Omron CX-Programmer project 新工程 (CX-Programmer 9.50)

# PLC 新PLC1: CP1H XA

## Global symbols (name address type ; comment)
0.01 BOOL  ; 启动
0.02 BOOL  ; 停止
0.04 BOOL  ; 急停
0.05 BOOL  ; 相序保护
0.11 BOOL  ; 空压机热保护
100.03 BOOL  ; A平
100.04 BOOL  ; B平
100.05 BOOL  ; C平
100.06 BOOL  ; A进
100.07 BOOL  ; B进
101.00 BOOL  ; C进
101.01 BOOL  ; A排
101.02 BOOL  ; b排
101.03 BOOL  ; C排
10.00 BOOL  ; 连续与自动
200 CHANNEL  ; 氧气纯度
201 CHANNEL  ; 空气压力
202 CHANNEL  ; 氧气压力
203 CHANNEL  ; 露点
A526.01 BOOL  ; 串行端口1重启标志
A528.11 BOOL  ; 出错标志
D1 CHANNEL  ; 空气压力上限
D10 CHANNEL  ; 屏显露点
D11 CHANNEL  ; 屏显氧气压力
D12 CHANNEL  ; 屏输空气压力下限
D13 CHANNEL  ; 屏显油温
D15 CHANNEL  ; 屏输空气压力上限
D17 CHANNEL  ; 屏输空气压力下限
D19 CHANNEL  ; 屏输氧气压力上限
D2 CHANNEL  ; 空气压力下限
D20 CHANNEL  ; 制氧机工作状态
D21 CHANNEL  ; 屏输氧气压力下限
D3 CHANNEL  ; 氧气压力上限
D3102 CHANNEL  ; 流量高位
D3103 CHANNEL  ; 流量低位
D3104 CHANNEL  ; 总流量高位
D3105 CHANNEL  ; 总流量低位
D317 CHANNEL  ; 制氧机状态字
D318 CHANNEL  ; 冷干机状态字
D321 CHANNEL  ; 系统状态字
D331 CHANNEL  ; 空压机状态字
D332 CHANNEL  ; 空滤维保计时
D333 CHANNEL  ; 油滤维保计时
D334 CHANNEL  ; 油分维保计时
D335 CHANNEL  ; 机油维保计时
D336 CHANNEL  ; 管滤维保计时
D337 CHANNEL  ; 菌滤维保计时
D338 CHANNEL  ; 制氧机工作状态
D4 CHANNEL  ; 氧气压力下限
D50 CHANNEL  ; 瞬时流量
D51 CHANNEL  ; 瞬时流量
D65 CHANNEL  ; 氧气压力
D66 CHANNEL  ; 空气压力
D67 CHANNEL  ; 油温
D68 CHANNEL  ; 氧气纯度
D69 CHANNEL  ; 氧气流量
D7 CHANNEL  ; 屏显氧气纯度
D8 CHANNEL  ; 屏显空气压力
D80 CHANNEL  ; 远程氧气
D82 CHANNEL  ; 远程空气
D84 CHANNEL  ; 远程油温
D86 CHANNEL  ; 远程氧气纯度
D88 CHANNEL  ; 远程氧气流量
D9 CHANNEL  ; 屏显空气压力
H1 CHANNEL  ; 运行总时间
H10.00 BOOL  ; 远程控制停机（保持）
H2 CHANNEL  ; 空滤维保计时
H3 CHANNEL  ; 油滤维保计时
H4 CHANNEL  ; 油分维保计时
H5 CHANNEL  ; 机油维保计时
H6 CHANNEL  ; 管滤维保计时
H7 CHANNEL  ; 菌滤维保计时
T0200 BOOL  ; 产生0.2秒脉冲
W10.00 BOOL  ; 连续与自动
W21.00 BOOL  ; 启动标志1
W21.01 BOOL  ; 散热见机
W21.02 BOOL  ; 外接排风
W21.03 BOOL  ; 冷干机
W21.04 BOOL  ; 卸载电磁阀
W21.05 BOOL  ; 空压机
W21.06 BOOL  ; 油温开关
W21.08 BOOL  ; 运行标志
W21.09 BOOL  ; 停机保护2分钟
W21.10 BOOL  ; 启动标志2
W21.11 BOOL  ; 出氧电磁阀
W21.12 BOOL  ; 准备待机
W21.13 BOOL  ; 待机
W21.14 BOOL  ; 复位几个启动时间
W21.15 BOOL  ; 解除几个停机时间
W22.01 BOOL  ; 连续与自动
W22.06 BOOL  ; 油温开关
W23.00 BOOL  ; 制氧启动最低空气压力
W24.01 BOOL  ; 准备停机
W24.07 BOOL  ; 停机
W25.00 BOOL  ; 报警器
W30 CHANNEL  ; 屏显氧气纯度
W32.00 BOOL  ; 散热风机热保护
W32.01 BOOL  ; 报警解除
W50.01 BOOL  ; 空滤维保复位
W50.02 BOOL  ; 油滤维保复位
W50.03 BOOL  ; 油分维保复位
W50.04 BOOL  ; 机油维保复位
W50.05 BOOL  ; 管滤维保复位
W50.06 BOOL  ; 菌滤维保复位
W50.15 BOOL  ; 躲开开机时氧气压力低
W8 CHANNEL  ; 计数器值

## Program 新程序1 (cyclic task 0)
Local symbols
Dd112 UINT
Dd300 UINT_BCD
P_0_6s BOOL
P_2分钟 BOOL
P_30分钟 BOOL
W BOOL
b189 UINT
ffff UINT

### Section 启动停止

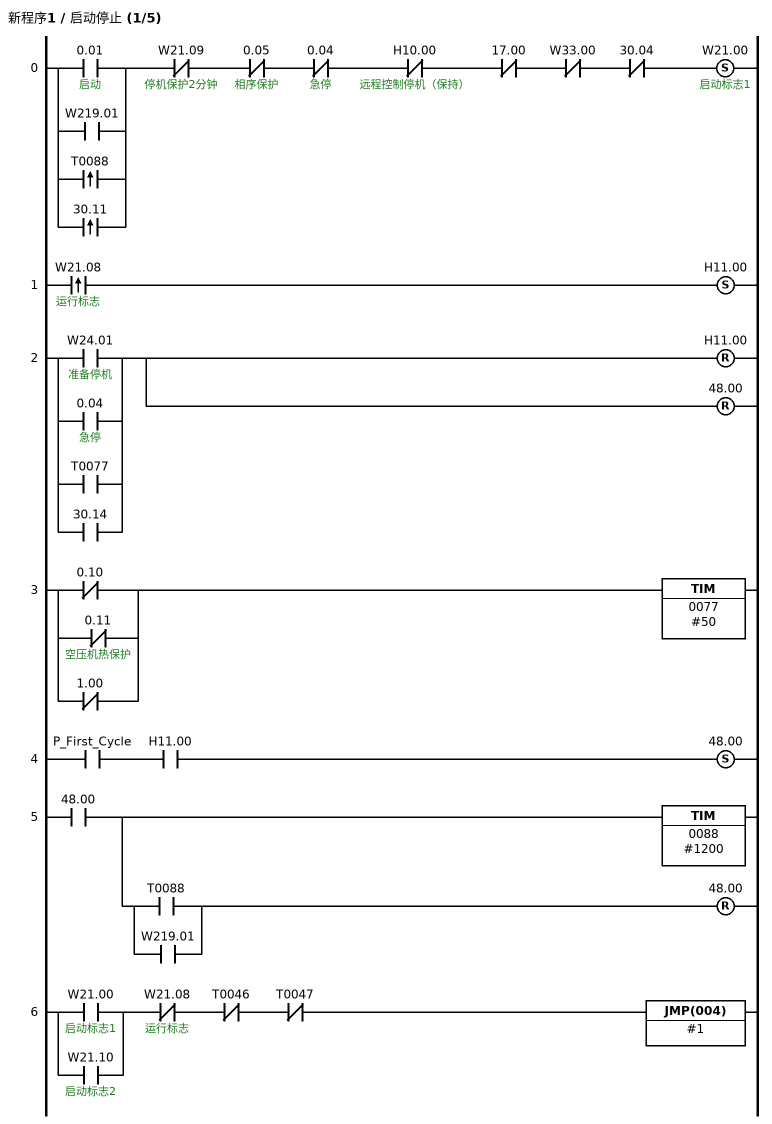
; rung 0
LD 0.01  ; 启动
OR W219.01
@OR T0088
@OR 30.11
ANDNOT W21.09  ; 停机保护2分钟
ANDNOT 0.05  ; 相序保护
ANDNOT 0.04  ; 急停
ANDNOT H10.00  ; 远程控制停机（保持）
ANDNOT 17.00
ANDNOT W33.00
ANDNOT 30.04
SET W21.00  ; 启动标志1
; rung 1
@LD W21.08  ; 运行标志
SET H11.00
; rung 2
LD W24.01  ; 准备停机
OR 0.04  ; 急停
OR T0077
OR 30.14
RSET H11.00
RSET 48.00
; rung 3
LDNOT 0.10
ORNOT 0.11  ; 空压机热保护
ORNOT 1.00
TIM 0077 #50
; rung 4
LD P_First_Cycle
AND H11.00
SET 48.00
; rung 5
LD 48.00
TIM 0088 #1200
LD T0088
OR W219.01
ANDLD
RSET 48.00
; rung 6
LD W21.00  ; 启动标志1
OR W21.10  ; 启动标志2
ANDNOT W21.08  ; 运行标志
ANDNOT T0046
ANDNOT T0047
JMP(004) #1

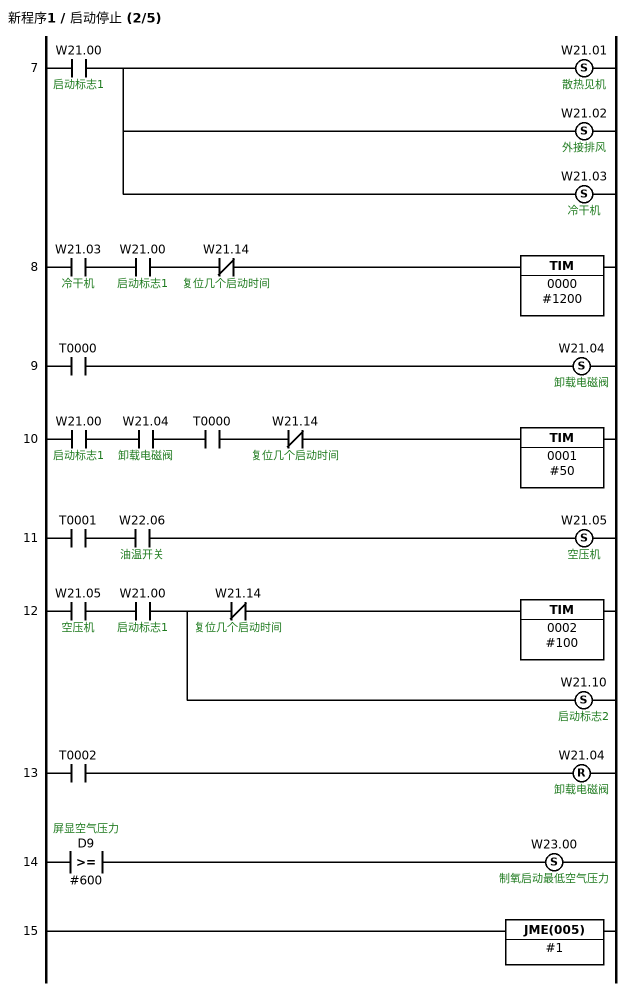
; rung 7
LD W21.00  ; 启动标志1
SET W21.01  ; 散热见机
SET W21.02  ; 外接排风
SET W21.03  ; 冷干机
; rung 8
LD W21.03  ; 冷干机
AND W21.00  ; 启动标志1
ANDNOT W21.14  ; 复位几个启动时间
TIM 0000 #1200
; rung 9
LD T0000
SET W21.04  ; 卸载电磁阀
; rung 10
LD W21.00  ; 启动标志1
AND W21.04  ; 卸载电磁阀
AND T0000
ANDNOT W21.14  ; 复位几个启动时间
TIM 0001 #50
; rung 11
LD T0001
AND W22.06  ; 油温开关
SET W21.05  ; 空压机
; rung 12
LD W21.05  ; 空压机
AND W21.00  ; 启动标志1
OUT TR0
ANDNOT W21.14  ; 复位几个启动时间
TIM 0002 #100
LD TR0
SET W21.10  ; 启动标志2
; rung 13
LD T0002
RSET W21.04  ; 卸载电磁阀
; rung 14
LD>=(325) D9 #600  ; 屏显空气压力
SET W23.00  ; 制氧启动最低空气压力
; rung 15
JME(005) #1

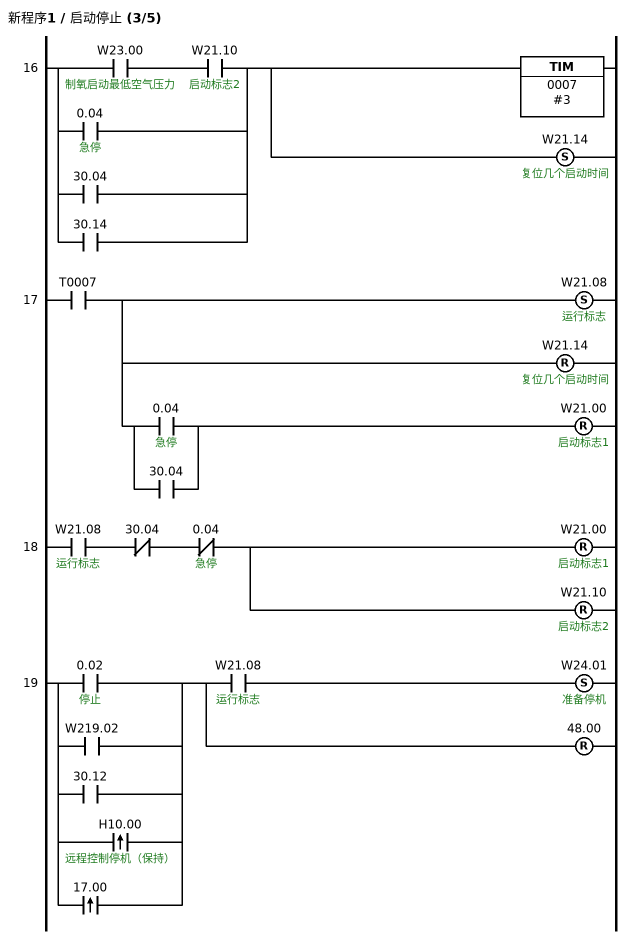
; rung 16
LD W23.00  ; 制氧启动最低空气压力
AND W21.10  ; 启动标志2
OR 0.04  ; 急停
OR 30.04
OR 30.14
TIM 0007 #3
SET W21.14  ; 复位几个启动时间
; rung 17
LD T0007
SET W21.08  ; 运行标志
RSET W21.14  ; 复位几个启动时间
LD 0.04  ; 急停
OR 30.04
ANDLD
RSET W21.00  ; 启动标志1
; rung 18
LD W21.08  ; 运行标志
ANDNOT 30.04
ANDNOT 0.04  ; 急停
RSET W21.00  ; 启动标志1
RSET W21.10  ; 启动标志2
; rung 19
LD 0.02  ; 停止
OR W219.02
OR 30.12
@OR H10.00  ; 远程控制停机（保持）
@OR 17.00
OUT TR0
AND W21.08  ; 运行标志
SET W24.01  ; 准备停机
LD TR0
RSET 48.00

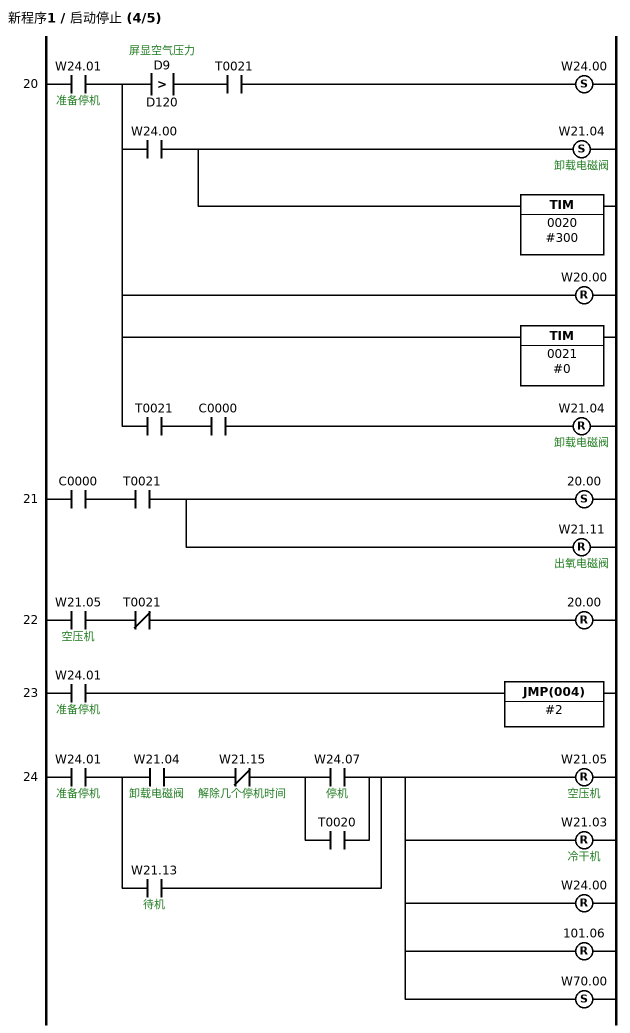
; rung 20
LD W24.01  ; 准备停机
OUT TR0
AND>(320) D9 D120  ; 屏显空气压力
AND T0021
SET W24.00
LD TR0
AND W24.00
SET W21.04  ; 卸载电磁阀
TIM 0020 #300
LD TR0
RSET W20.00
TIM 0021 #0
AND T0021
AND C0000
RSET W21.04  ; 卸载电磁阀
; rung 21
LD C0000
AND T0021
SET 20.00
RSET W21.11  ; 出氧电磁阀
; rung 22
LD W21.05  ; 空压机
ANDNOT T0021
RSET 20.00
; rung 23
LD W24.01  ; 准备停机
JMP(004) #2
; rung 24
LD W24.01  ; 准备停机
LD W21.04  ; 卸载电磁阀
ANDNOT W21.15  ; 解除几个停机时间
LD W24.07  ; 停机
OR T0020
ANDLD
OR W21.13  ; 待机
ANDLD
RSET W21.05  ; 空压机
RSET W21.03  ; 冷干机
RSET W24.00
RSET 101.06
SET W70.00

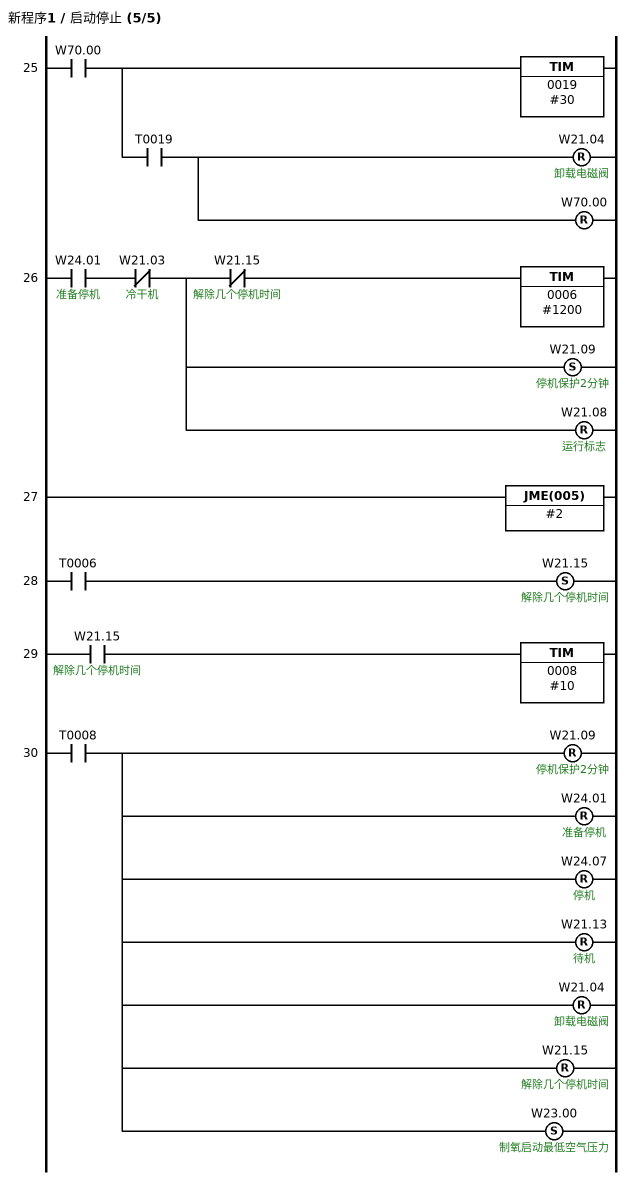
; rung 25
LD W70.00
TIM 0019 #30
AND T0019
RSET W21.04  ; 卸载电磁阀
RSET W70.00
; rung 26
LD W24.01  ; 准备停机
ANDNOT W21.03  ; 冷干机
OUT TR0
ANDNOT W21.15  ; 解除几个停机时间
TIM 0006 #1200
LD TR0
SET W21.09  ; 停机保护2分钟
RSET W21.08  ; 运行标志
; rung 27
JME(005) #2
; rung 28
LD T0006
SET W21.15  ; 解除几个停机时间
; rung 29
LD W21.15  ; 解除几个停机时间
TIM 0008 #10
; rung 30
LD T0008
RSET W21.09  ; 停机保护2分钟
RSET W24.01  ; 准备停机
RSET W24.07  ; 停机
RSET W21.13  ; 待机
RSET W21.04  ; 卸载电磁阀
RSET W21.15  ; 解除几个停机时间
SET W23.00  ; 制氧启动最低空气压力

### Section 制氧机时间

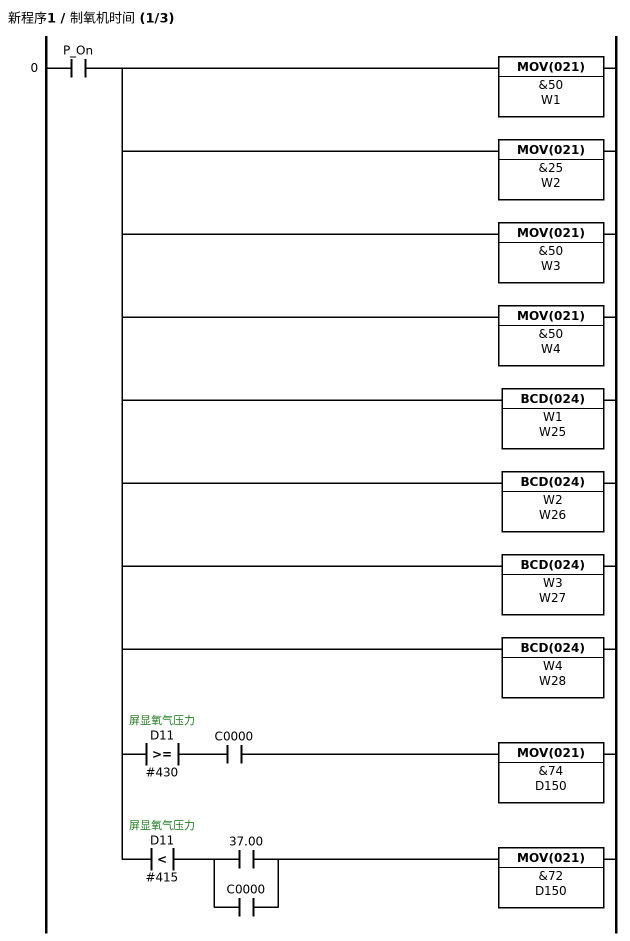
; rung 0
LD P_On
OUT TR0
MOV(021) &50 W1
MOV(021) &25 W2
MOV(021) &50 W3
MOV(021) &50 W4
BCD(024) W1 W25
BCD(024) W2 W26
BCD(024) W3 W27
BCD(024) W4 W28
AND>=(325) D11 #430  ; 屏显氧气压力
AND C0000
MOV(021) &74 D150
LD TR0
AND<(310) D11 #415  ; 屏显氧气压力
LD 37.00
OR C0000
ANDLD
MOV(021) &72 D150

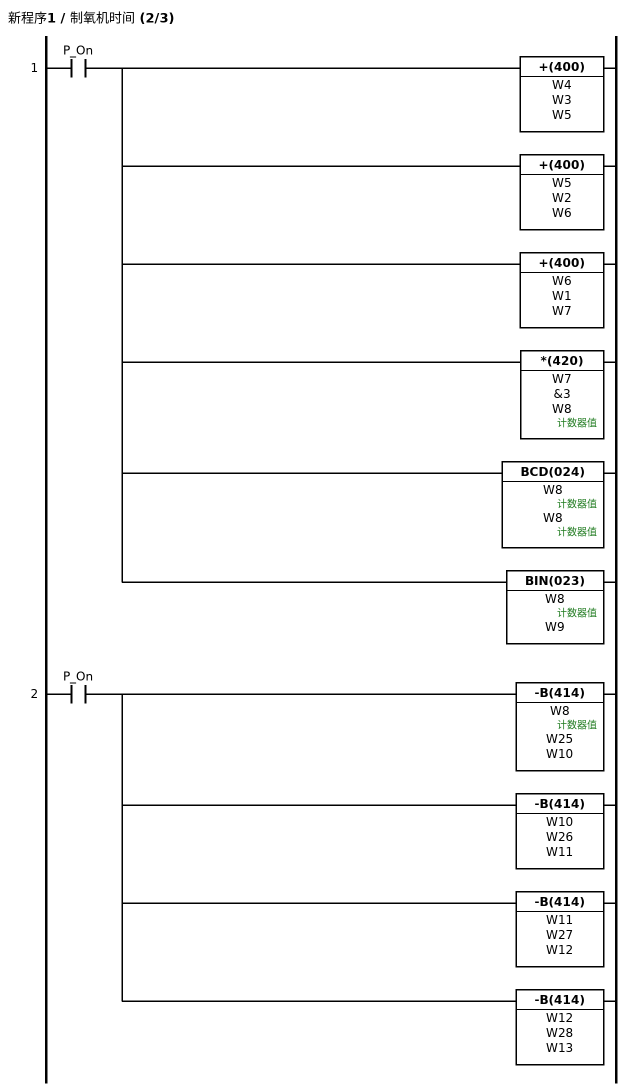
; rung 1
LD P_On
+(400) W4 W3 W5
+(400) W5 W2 W6
+(400) W6 W1 W7
*(420) W7 &3 W8  ; 计数器值
BCD(024) W8 W8  ; 计数器值
BIN(023) W8 W9  ; 计数器值
; rung 2
LD P_On
-B(414) W8 W25 W10  ; 计数器值
-B(414) W10 W26 W11
-B(414) W11 W27 W12
-B(414) W12 W28 W13

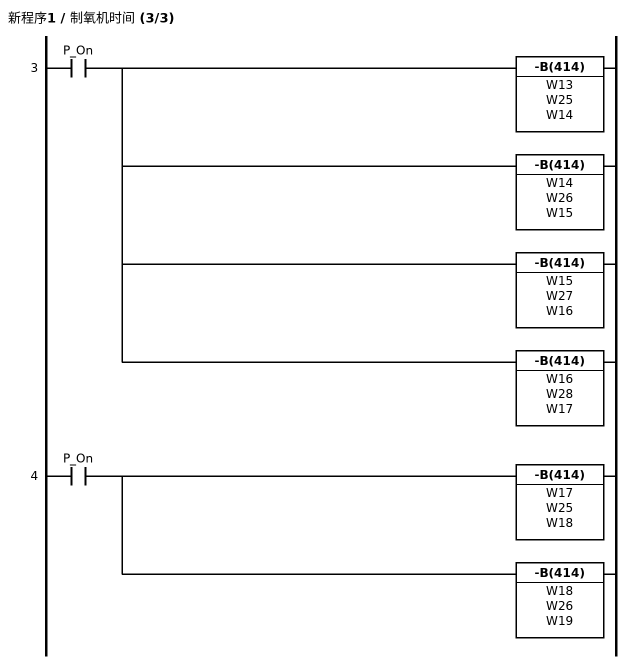
; rung 3
LD P_On
-B(414) W13 W25 W14
-B(414) W14 W26 W15
-B(414) W15 W27 W16
-B(414) W16 W28 W17
; rung 4
LD P_On
-B(414) W17 W25 W18
-B(414) W18 W26 W19

### Section 制氧机步骤

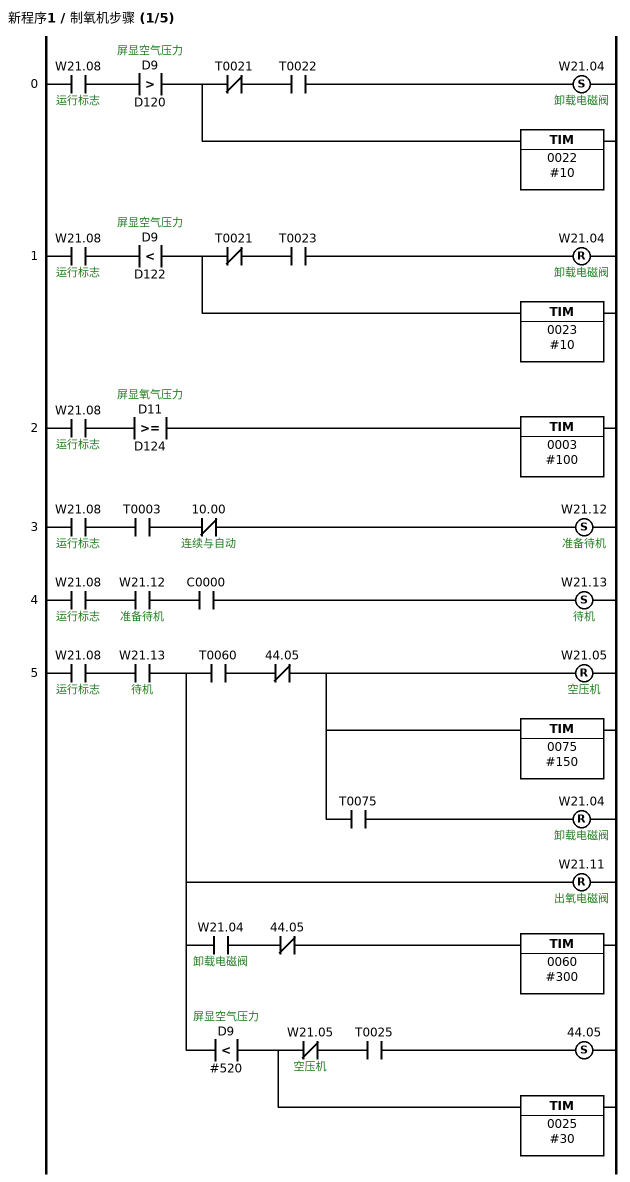
; rung 0
LD W21.08  ; 运行标志
AND>(320) D9 D120  ; 屏显空气压力
OUT TR0
ANDNOT T0021
AND T0022
SET W21.04  ; 卸载电磁阀
LD TR0
TIM 0022 #10
; rung 1
LD W21.08  ; 运行标志
AND<(310) D9 D122  ; 屏显空气压力
OUT TR0
ANDNOT T0021
AND T0023
RSET W21.04  ; 卸载电磁阀
LD TR0
TIM 0023 #10
; rung 2
LD W21.08  ; 运行标志
AND>=(325) D11 D124  ; 屏显氧气压力
TIM 0003 #100
; rung 3
LD W21.08  ; 运行标志
AND T0003
ANDNOT 10.00  ; 连续与自动
SET W21.12  ; 准备待机
; rung 4
LD W21.08  ; 运行标志
AND W21.12  ; 准备待机
AND C0000
SET W21.13  ; 待机
; rung 5
LD W21.08  ; 运行标志
AND W21.13  ; 待机
OUT TR0
AND T0060
ANDNOT 44.05
RSET W21.05  ; 空压机
TIM 0075 #150
AND T0075
RSET W21.04  ; 卸载电磁阀
LD TR0
RSET W21.11  ; 出氧电磁阀
AND W21.04  ; 卸载电磁阀
ANDNOT 44.05
TIM 0060 #300
LD TR0
AND<(310) D9 #520  ; 屏显空气压力
OUT TR0
ANDNOT W21.05  ; 空压机
AND T0025
SET 44.05
LD TR0
TIM 0025 #30

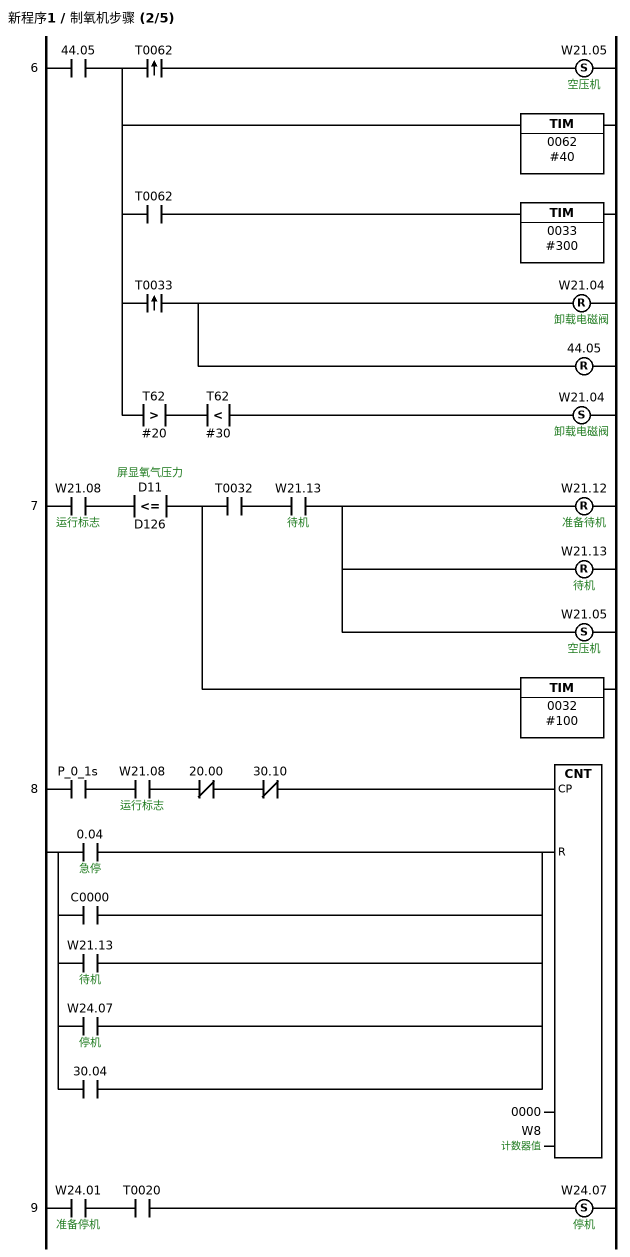
; rung 6
LD 44.05
OUT TR0
@AND T0062
SET W21.05  ; 空压机
LD TR0
TIM 0062 #40
AND T0062
TIM 0033 #300
LD TR0
@AND T0033
RSET W21.04  ; 卸载电磁阀
RSET 44.05
LD TR0
AND>(320) T62 #20
AND<(310) T62 #30
SET W21.04  ; 卸载电磁阀
; rung 7
LD W21.08  ; 运行标志
AND<=(315) D11 D126  ; 屏显氧气压力
OUT TR0
AND T0032
AND W21.13  ; 待机
RSET W21.12  ; 准备待机
RSET W21.13  ; 待机
SET W21.05  ; 空压机
LD TR0
TIM 0032 #100
; rung 8
LD P_0_1s
AND W21.08  ; 运行标志
ANDNOT 20.00
ANDNOT 30.10
LD 0.04  ; 急停
OR C0000
OR W21.13  ; 待机
OR W24.07  ; 停机
OR 30.04
CNT 0000 W8  ; 计数器值
; rung 9
LD W24.01  ; 准备停机
AND T0020
SET W24.07  ; 停机

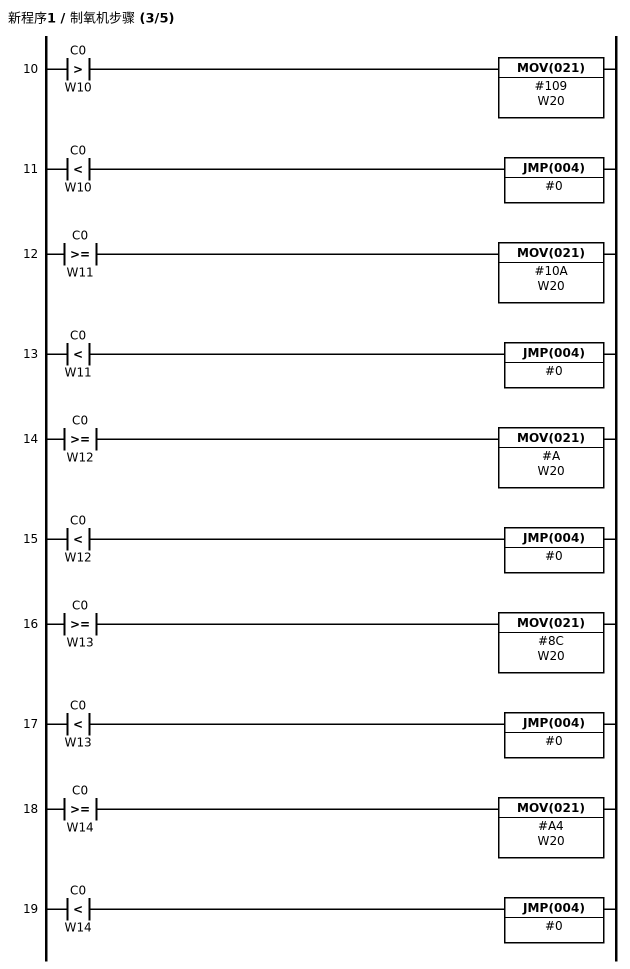
; rung 10
LD>(320) C0 W10
MOV(021) #109 W20
; rung 11
LD<(310) C0 W10
JMP(004) #0
; rung 12
LD>=(325) C0 W11
MOV(021) #10A W20
; rung 13
LD<(310) C0 W11
JMP(004) #0
; rung 14
LD>=(325) C0 W12
MOV(021) #A W20
; rung 15
LD<(310) C0 W12
JMP(004) #0
; rung 16
LD>=(325) C0 W13
MOV(021) #8C W20
; rung 17
LD<(310) C0 W13
JMP(004) #0
; rung 18
LD>=(325) C0 W14
MOV(021) #A4 W20
; rung 19
LD<(310) C0 W14
JMP(004) #0

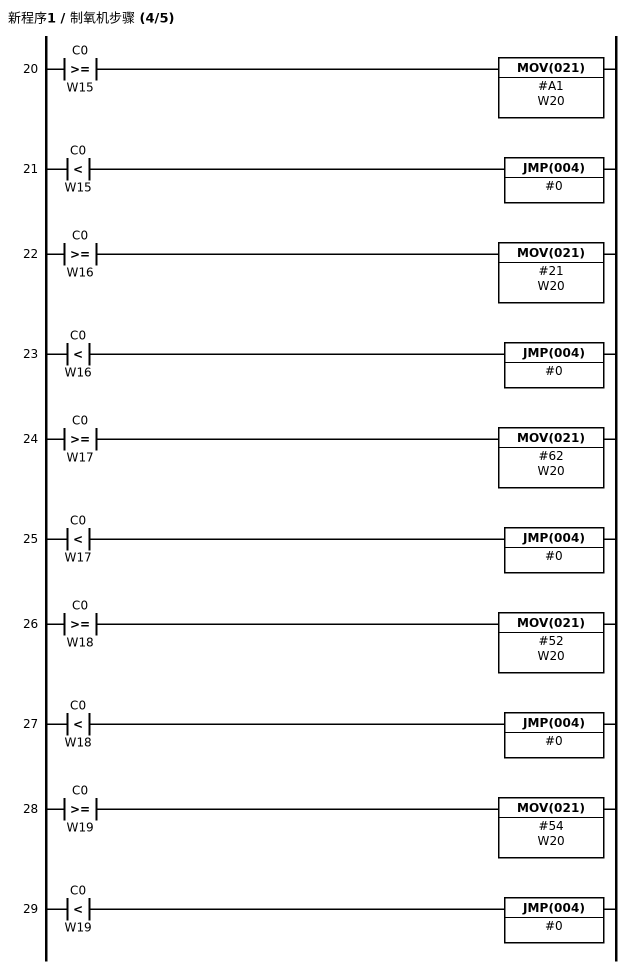
; rung 20
LD>=(325) C0 W15
MOV(021) #A1 W20
; rung 21
LD<(310) C0 W15
JMP(004) #0
; rung 22
LD>=(325) C0 W16
MOV(021) #21 W20
; rung 23
LD<(310) C0 W16
JMP(004) #0
; rung 24
LD>=(325) C0 W17
MOV(021) #62 W20
; rung 25
LD<(310) C0 W17
JMP(004) #0
; rung 26
LD>=(325) C0 W18
MOV(021) #52 W20
; rung 27
LD<(310) C0 W18
JMP(004) #0
; rung 28
LD>=(325) C0 W19
MOV(021) #54 W20
; rung 29
LD<(310) C0 W19
JMP(004) #0

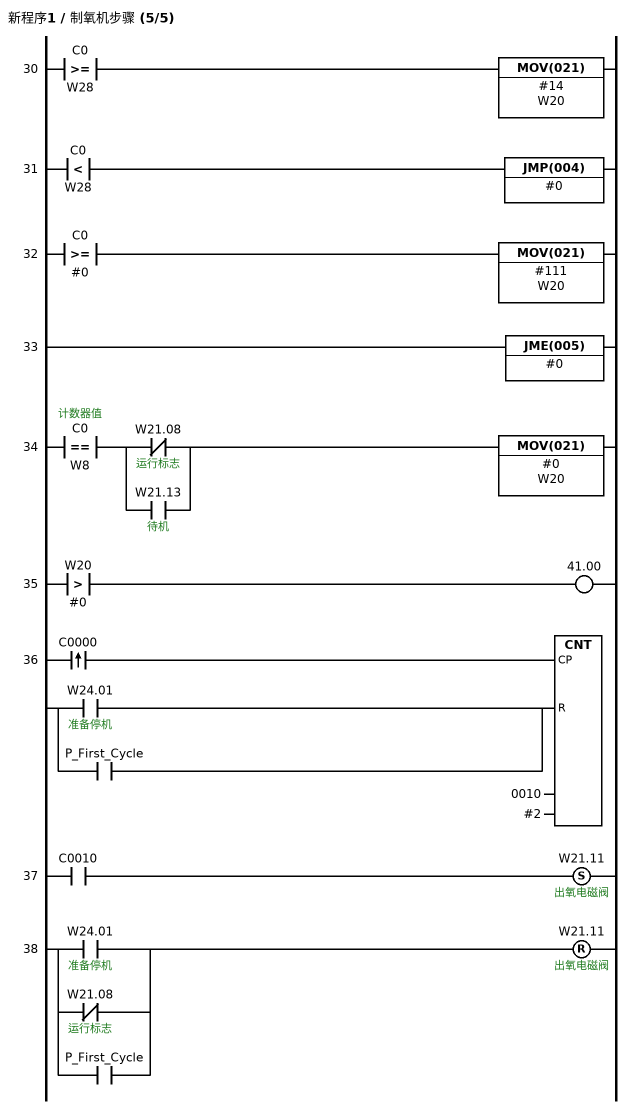
; rung 30
LD>=(325) C0 W28
MOV(021) #14 W20
; rung 31
LD<(310) C0 W28
JMP(004) #0
; rung 32
LD>=(325) C0 #0
MOV(021) #111 W20
; rung 33
JME(005) #0
; rung 34
LD=(300) C0 W8  ; 计数器值
LDNOT W21.08  ; 运行标志
OR W21.13  ; 待机
ANDLD
MOV(021) #0 W20
; rung 35
LD>(320) W20 #0
OUT 41.00
; rung 36
@LD C0000
LD W24.01  ; 准备停机
OR P_First_Cycle
CNT 0010 #2
; rung 37
LD C0010
SET W21.11  ; 出氧电磁阀
; rung 38
LD W24.01  ; 准备停机
ORNOT W21.08  ; 运行标志
OR P_First_Cycle
RSET W21.11  ; 出氧电磁阀

### Section _4AD数值

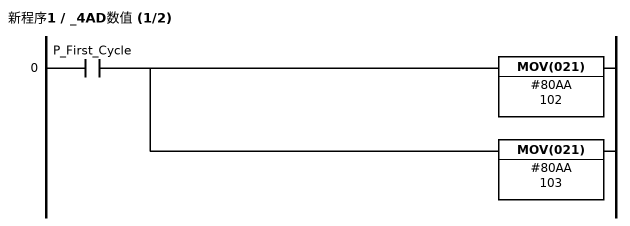
; rung 0
LD P_First_Cycle
MOV(021) #80AA 102
MOV(021) #80AA 103

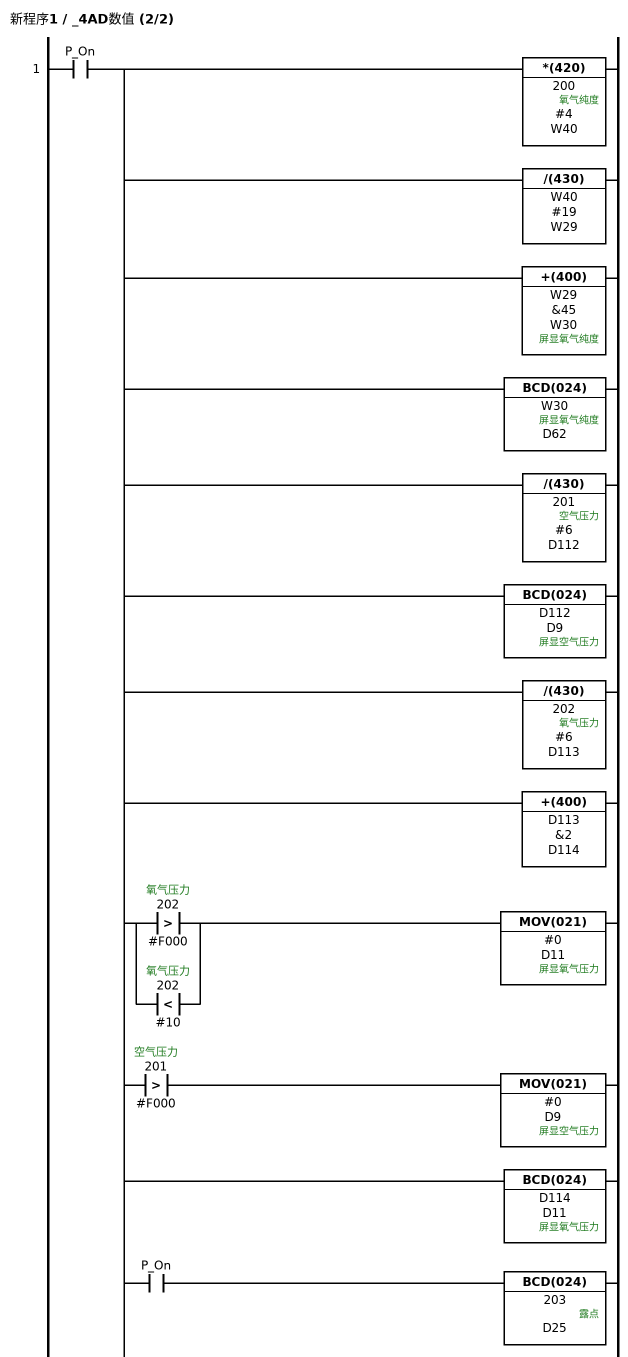

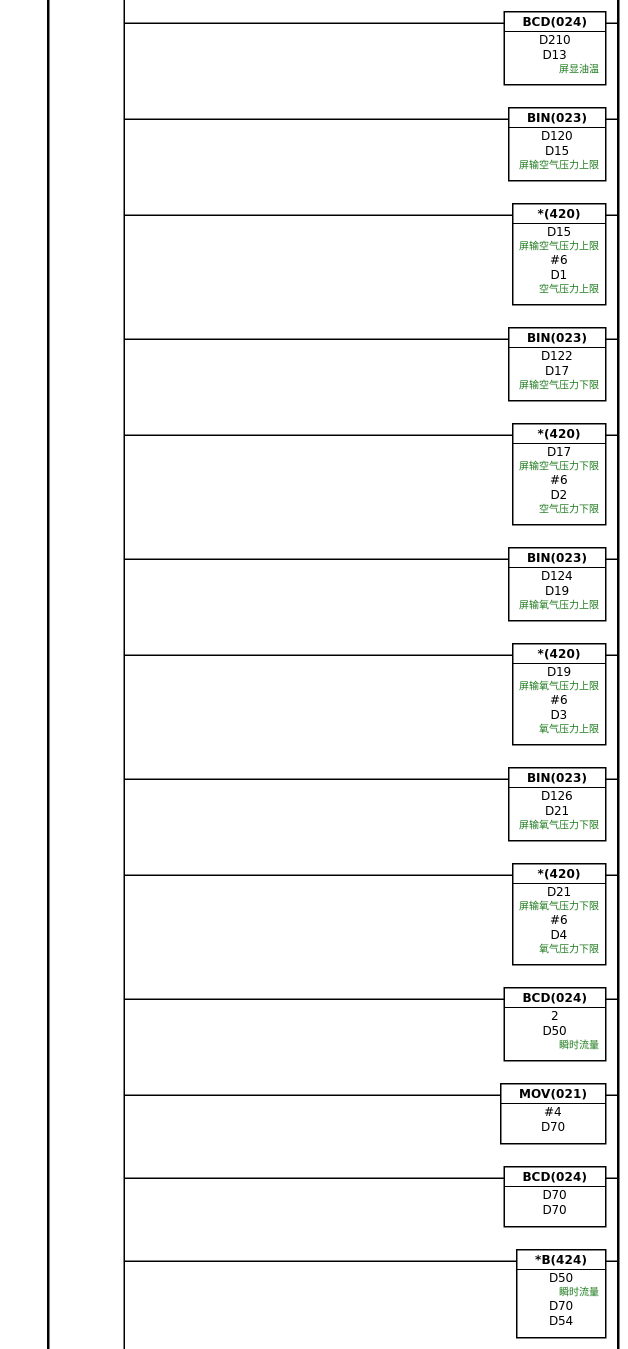

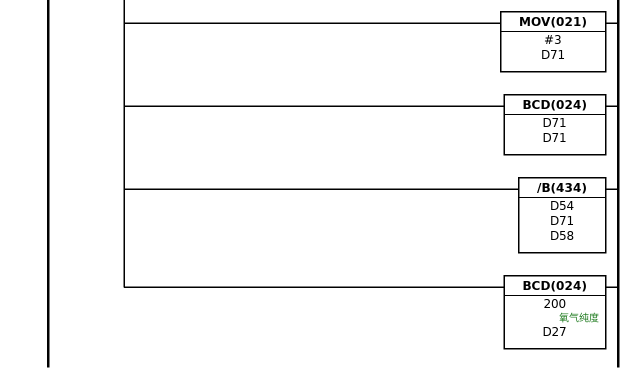
; rung 1
LD P_On
OUT TR0
*(420) 200 #4 W40  ; 氧气纯度
/(430) W40 #19 W29
+(400) W29 &45 W30  ; 屏显氧气纯度
BCD(024) W30 D62  ; 屏显氧气纯度
/(430) 201 #6 D112  ; 空气压力
BCD(024) D112 D9  ; 屏显空气压力
/(430) 202 #6 D113  ; 氧气压力
+(400) D113 &2 D114
LD>(320) 202 #F000  ; 氧气压力
OR<(310) 202 #10  ; 氧气压力
ANDLD
MOV(021) #0 D11  ; 屏显氧气压力
LD TR0
AND>(320) 201 #F000  ; 空气压力
MOV(021) #0 D9  ; 屏显空气压力
LD TR0
BCD(024) D114 D11  ; 屏显氧气压力
AND P_On
BCD(024) 203 D25  ; 露点
LD TR0
BCD(024) D210 D13  ; 屏显油温
BIN(023) D120 D15  ; 屏输空气压力上限
*(420) D15 #6 D1  ; 屏输空气压力上限, 空气压力上限
BIN(023) D122 D17  ; 屏输空气压力下限
*(420) D17 #6 D2  ; 屏输空气压力下限, 空气压力下限
BIN(023) D124 D19  ; 屏输氧气压力上限
*(420) D19 #6 D3  ; 屏输氧气压力上限, 氧气压力上限
BIN(023) D126 D21  ; 屏输氧气压力下限
*(420) D21 #6 D4  ; 屏输氧气压力下限, 氧气压力下限
BCD(024) 2 D50  ; 瞬时流量
MOV(021) #4 D70
BCD(024) D70 D70
*B(424) D50 D70 D54  ; 瞬时流量
MOV(021) #3 D71
BCD(024) D71 D71
/B(434) D54 D71 D58
BCD(024) 200 D27  ; 氧气纯度

### Section 报警耗材设定

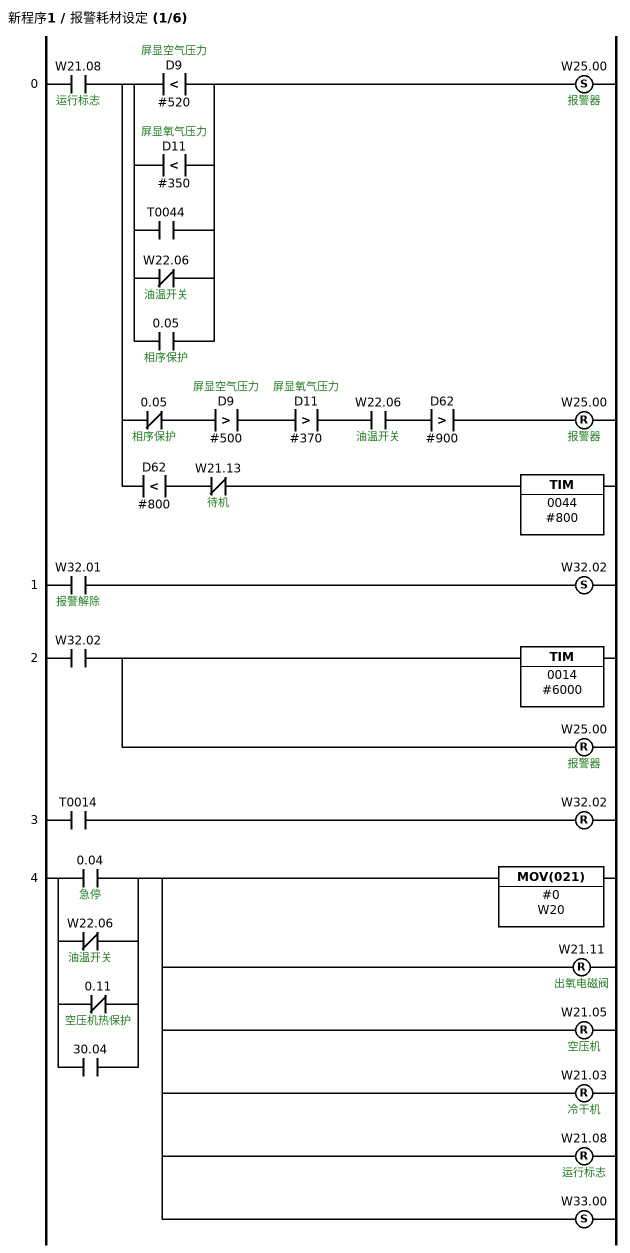
; rung 0
LD W21.08  ; 运行标志
OUT TR0
LD<(310) D9 #520  ; 屏显空气压力
OR<(310) D11 #350  ; 屏显氧气压力
OR T0044
ORNOT W22.06  ; 油温开关
OR 0.05  ; 相序保护
ANDLD
SET W25.00  ; 报警器
LD TR0
ANDNOT 0.05  ; 相序保护
AND>(320) D9 #500  ; 屏显空气压力
AND>(320) D11 #370  ; 屏显氧气压力
AND W22.06  ; 油温开关
AND>(320) D62 #900
RSET W25.00  ; 报警器
LD TR0
AND<(310) D62 #800
ANDNOT W21.13  ; 待机
TIM 0044 #800
; rung 1
LD W32.01  ; 报警解除
SET W32.02
; rung 2
LD W32.02
TIM 0014 #6000
RSET W25.00  ; 报警器
; rung 3
LD T0014
RSET W32.02
; rung 4
LD 0.04  ; 急停
ORNOT W22.06  ; 油温开关
ORNOT 0.11  ; 空压机热保护
OR 30.04
MOV(021) #0 W20
RSET W21.11  ; 出氧电磁阀
RSET W21.05  ; 空压机
RSET W21.03  ; 冷干机
RSET W21.08  ; 运行标志
SET W33.00

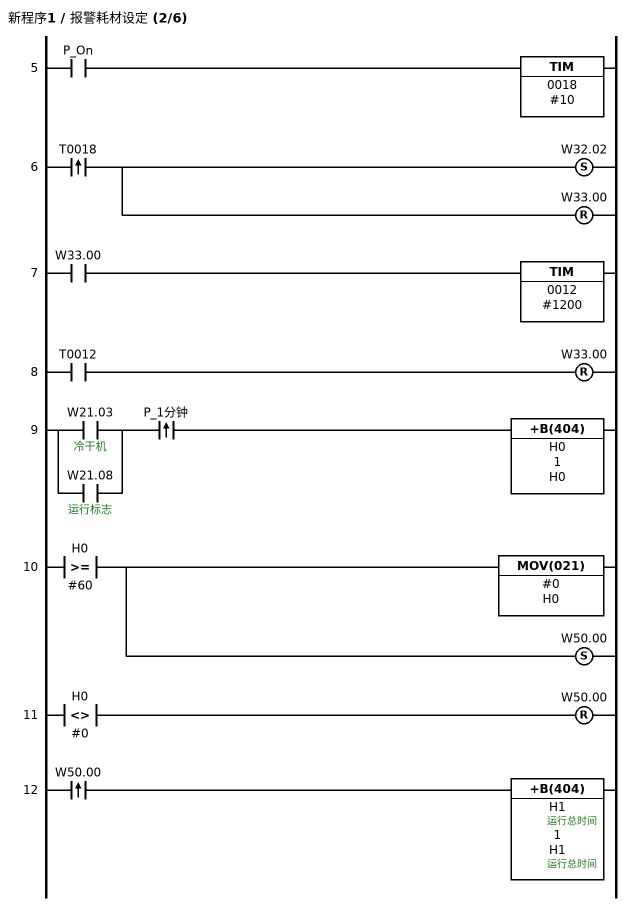
; rung 5
LD P_On
TIM 0018 #10
; rung 6
@LD T0018
SET W32.02
RSET W33.00
; rung 7
LD W33.00
TIM 0012 #1200
; rung 8
LD T0012
RSET W33.00
; rung 9
LD W21.03  ; 冷干机
OR W21.08  ; 运行标志
@AND P_1分钟
+B(404) H0 1 H0
; rung 10
LD>=(325) H0 #60
MOV(021) #0 H0
SET W50.00
; rung 11
LD<>(305) H0 #0
RSET W50.00
; rung 12
@LD W50.00
+B(404) H1 1 H1  ; 运行总时间

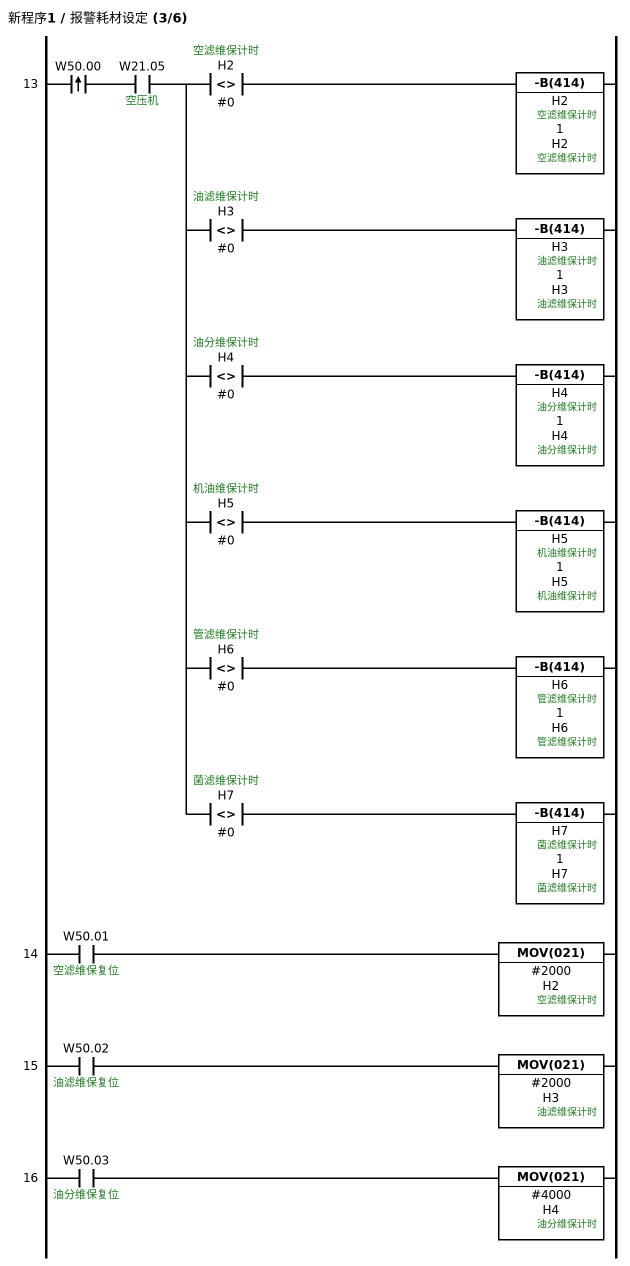
; rung 13
@LD W50.00
AND W21.05  ; 空压机
OUT TR0
AND<>(305) H2 #0  ; 空滤维保计时
-B(414) H2 1 H2  ; 空滤维保计时
LD TR0
AND<>(305) H3 #0  ; 油滤维保计时
-B(414) H3 1 H3  ; 油滤维保计时
LD TR0
AND<>(305) H4 #0  ; 油分维保计时
-B(414) H4 1 H4  ; 油分维保计时
LD TR0
AND<>(305) H5 #0  ; 机油维保计时
-B(414) H5 1 H5  ; 机油维保计时
LD TR0
AND<>(305) H6 #0  ; 管滤维保计时
-B(414) H6 1 H6  ; 管滤维保计时
LD TR0
AND<>(305) H7 #0  ; 菌滤维保计时
-B(414) H7 1 H7  ; 菌滤维保计时
; rung 14
LD W50.01  ; 空滤维保复位
MOV(021) #2000 H2  ; 空滤维保计时
; rung 15
LD W50.02  ; 油滤维保复位
MOV(021) #2000 H3  ; 油滤维保计时
; rung 16
LD W50.03  ; 油分维保复位
MOV(021) #4000 H4  ; 油分维保计时

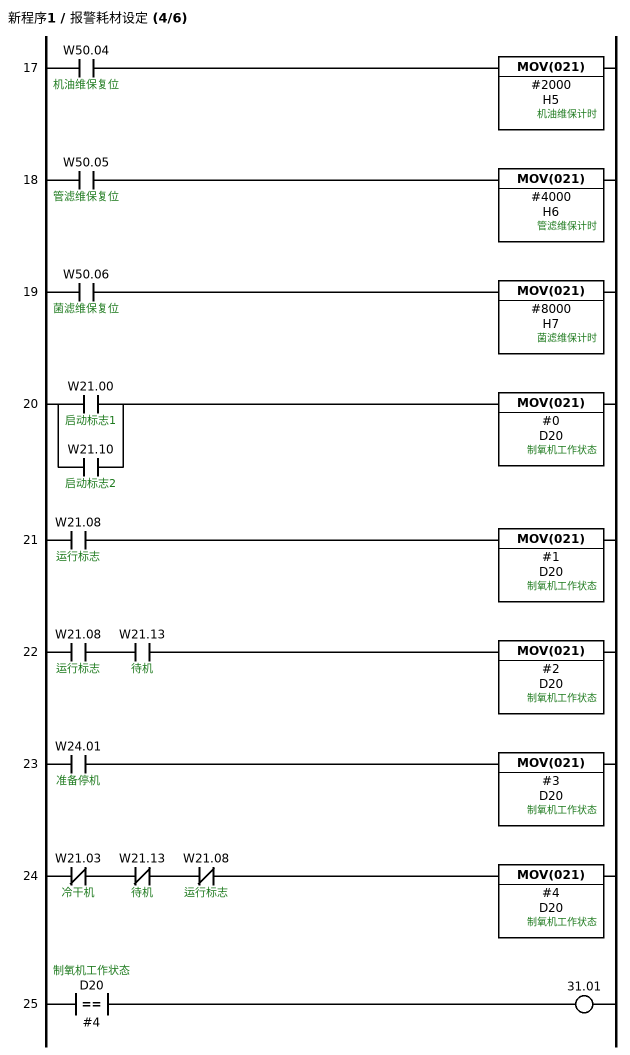
; rung 17
LD W50.04  ; 机油维保复位
MOV(021) #2000 H5  ; 机油维保计时
; rung 18
LD W50.05  ; 管滤维保复位
MOV(021) #4000 H6  ; 管滤维保计时
; rung 19
LD W50.06  ; 菌滤维保复位
MOV(021) #8000 H7  ; 菌滤维保计时
; rung 20
LD W21.00  ; 启动标志1
OR W21.10  ; 启动标志2
MOV(021) #0 D20  ; 制氧机工作状态
; rung 21
LD W21.08  ; 运行标志
MOV(021) #1 D20  ; 制氧机工作状态
; rung 22
LD W21.08  ; 运行标志
AND W21.13  ; 待机
MOV(021) #2 D20  ; 制氧机工作状态
; rung 23
LD W24.01  ; 准备停机
MOV(021) #3 D20  ; 制氧机工作状态
; rung 24
LDNOT W21.03  ; 冷干机
ANDNOT W21.13  ; 待机
ANDNOT W21.08  ; 运行标志
MOV(021) #4 D20  ; 制氧机工作状态
; rung 25
LD=(300) D20 #4  ; 制氧机工作状态
OUT 31.01

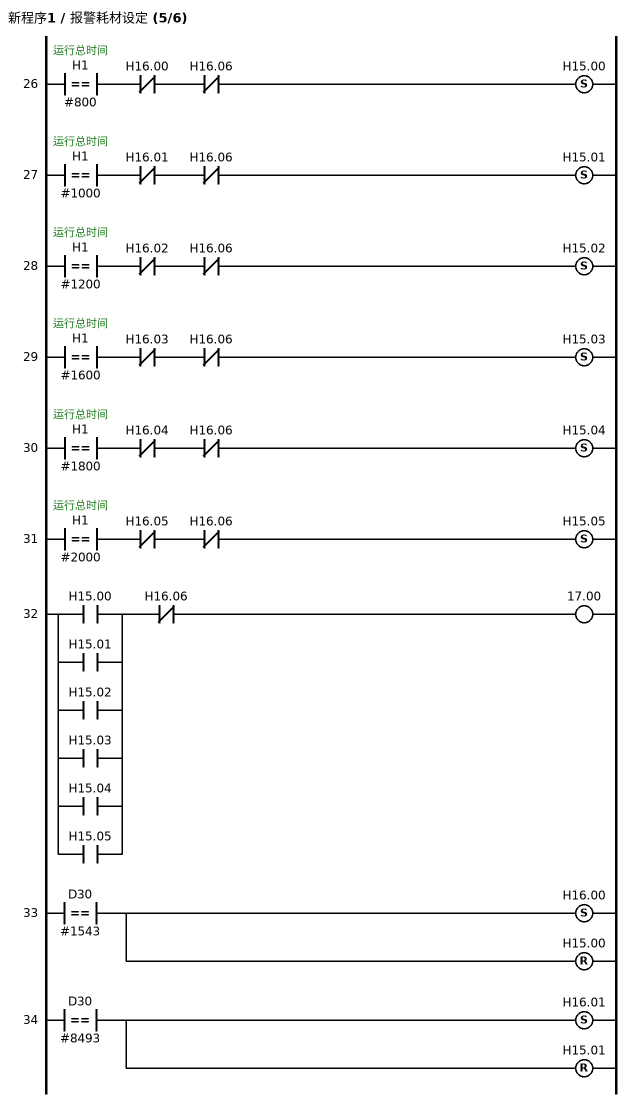
; rung 26
LD=(300) H1 #800  ; 运行总时间
ANDNOT H16.00
ANDNOT H16.06
SET H15.00
; rung 27
LD=(300) H1 #1000  ; 运行总时间
ANDNOT H16.01
ANDNOT H16.06
SET H15.01
; rung 28
LD=(300) H1 #1200  ; 运行总时间
ANDNOT H16.02
ANDNOT H16.06
SET H15.02
; rung 29
LD=(300) H1 #1600  ; 运行总时间
ANDNOT H16.03
ANDNOT H16.06
SET H15.03
; rung 30
LD=(300) H1 #1800  ; 运行总时间
ANDNOT H16.04
ANDNOT H16.06
SET H15.04
; rung 31
LD=(300) H1 #2000  ; 运行总时间
ANDNOT H16.05
ANDNOT H16.06
SET H15.05
; rung 32
LD H15.00
OR H15.01
OR H15.02
OR H15.03
OR H15.04
OR H15.05
ANDNOT H16.06
OUT 17.00
; rung 33
LD=(300) D30 #1543
SET H16.00
RSET H15.00
; rung 34
LD=(300) D30 #8493
SET H16.01
RSET H15.01

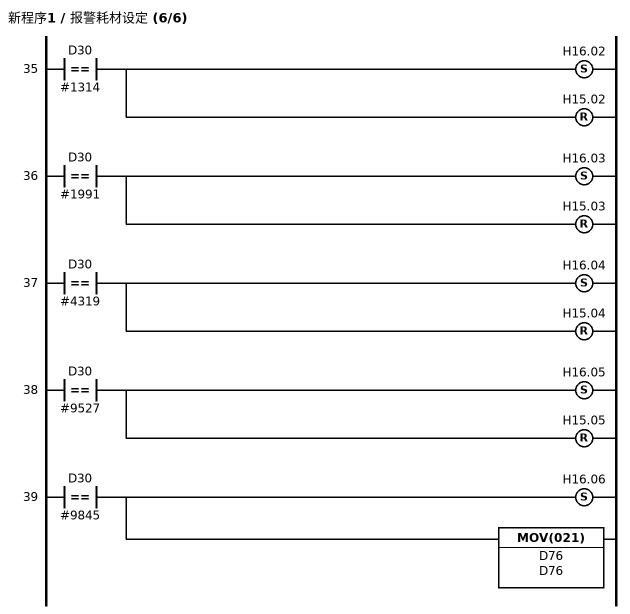
; rung 35
LD=(300) D30 #1314
SET H16.02
RSET H15.02
; rung 36
LD=(300) D30 #1991
SET H16.03
RSET H15.03
; rung 37
LD=(300) D30 #4319
SET H16.04
RSET H15.04
; rung 38
LD=(300) D30 #9527
SET H16.05
RSET H15.05
; rung 39
LD=(300) D30 #9845
SET H16.06
MOV(021) D76 D76

### Section 输出

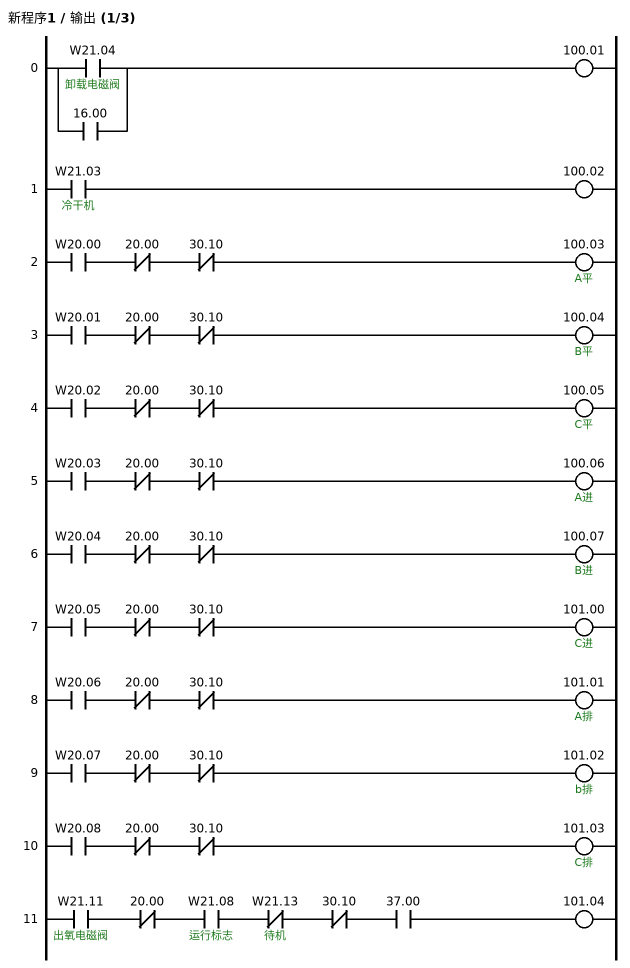
; rung 0
LD W21.04  ; 卸载电磁阀
OR 16.00
OUT 100.01
; rung 1
LD W21.03  ; 冷干机
OUT 100.02
; rung 2
LD W20.00
ANDNOT 20.00
ANDNOT 30.10
OUT 100.03  ; A平
; rung 3
LD W20.01
ANDNOT 20.00
ANDNOT 30.10
OUT 100.04  ; B平
; rung 4
LD W20.02
ANDNOT 20.00
ANDNOT 30.10
OUT 100.05  ; C平
; rung 5
LD W20.03
ANDNOT 20.00
ANDNOT 30.10
OUT 100.06  ; A进
; rung 6
LD W20.04
ANDNOT 20.00
ANDNOT 30.10
OUT 100.07  ; B进
; rung 7
LD W20.05
ANDNOT 20.00
ANDNOT 30.10
OUT 101.00  ; C进
; rung 8
LD W20.06
ANDNOT 20.00
ANDNOT 30.10
OUT 101.01  ; A排
; rung 9
LD W20.07
ANDNOT 20.00
ANDNOT 30.10
OUT 101.02  ; b排
; rung 10
LD W20.08
ANDNOT 20.00
ANDNOT 30.10
OUT 101.03  ; C排
; rung 11
LD W21.11  ; 出氧电磁阀
ANDNOT 20.00
AND W21.08  ; 运行标志
ANDNOT W21.13  ; 待机
ANDNOT 30.10
AND 37.00
OUT 101.04

